PROGRAM AnalogOutputEx
VAR
	fbHVACAnalogOutputEx: FB_HVACAnalogOutputEx;
	eDataSecurityType: E_HVACDataSecurityType := E_HVACDataSecurityType.eHVACDataSecurityType_Idle;
	bSetDefault: BOOL;
	bEnable: BOOL;
	rSetpoint: REAL;
	bCtrlVoltage: BOOL;
	eCtrlModeAnalogOutput: E_HVACAnalogOutputMode;
	rYManual: REAL;
	rFeedb: REAL;
	bFrost: BOOL;
	bReset: BOOL;
	rX2: REAL;
	rX1: REAL;
	iY2: INT;
	iY1: INT;
	bDirection: BOOL;
	bEnableFeedbCtrl: BOOL;
	rHysteresisFeedbCtrl: REAL;
	tDelayFeedbCtrl: TIME;
	rY: REAL;
	iYTerminal: INT;
	eStateModeAnalogOutput: Tc2_HVAC.E_HVACAnalogOutputMode;
	bManualMode: BOOL;
	byState: BYTE;
	bErrorFeedb: BOOL;
	bErrorGeneral: BOOL;
	byError: BYTE;
	bInvalidParameter: BOOL;
END_VAR

fbHVACAnalogOutputEx(
	eDataSecurityType:=eDataSecurityType, 
	bSetDefault:=bSetDefault, 
	bEnable:=bEnable, 
	rSetpoint:=rSetpoint, 
	bCtrlVoltage:=bCtrlVoltage, 
	eCtrlModeAnalogOutput:=eCtrlModeAnalogOutput, 
	rYManual:=rYManual, 
	rFeedb:=rFeedb, 
	bFrost:=bFrost, 
	bReset:=bReset, 
	rY=>rY, 
	iYTerminal=>iYTerminal, 
	eStateModeAnalogOutput=>eStateModeAnalogOutput, 
	bManualMode=>bManualMode, 
	byState=>byState, 
	bErrorFeedb=>bErrorFeedb, 
	bErrorGeneral=>bErrorGeneral, 
	byError=>byError, 
	bInvalidParameter=>bInvalidParameter, 
	rX2:=rX2, 
	rX1:=rX1, 
	iY2:=iY2, 
	iY1:=iY1, 
	bDirection:=bDirection, 
	bEnableFeedbCtrl:=bEnableFeedbCtrl, 
	rHysteresisFeedbCtrl:=rHysteresisFeedbCtrl, 
	tDelayFeedbCtrl:=tDelayFeedbCtrl);

END_PROGRAM

(* stored: Version 1.1.0.1, ProductVersion 3.1.4024.4
   POU AnalogOutputEx: Id {3de34637-d188-46b3-bf3f-7a94d0c8f3a9}, SpecialFunc None *)
